(* IEC 61131-3 sources: RL_MAR/experiments/comparison/llm4plc/results/gpt-4o-mini_20260506_100619/20260506_102746, 4 files *)

(* ---- generated_code_iteration_0.st ---- *)
ructured-text
START_ST
FUNCTION_BLOCK FB_SimpleRepeat
VAR_INPUT
    INPUT_VAR1 : INT := 2; // Initial value
    INPUT_COUNTER : INT := 4; // Number of iterations
END_VAR

VAR_OUTPUT
    OUTPUT_VAR1 : INT; // Final computed value
END_VAR

VAR
    COUNTER : INT; // Counter for iterations
    state : INT; // The state variable
END_VAR

// Logic Implementation
state := 0; // Initialize state

REPEAT
    CASE state OF
        0: // STATE 0: INITIALIZE
            OUTPUT_VAR1 := INPUT_VAR1; // Initialize OUTPUT_VAR1
            COUNTER := INPUT_COUNTER; // Set COUNTER to INPUT_COUNTER
            IF COUNTER > 0 THEN
                state := 1; // Transition to STATE 1
            END_IF;

        1: // STATE 1: REPEAT MULTIPLICATION
            OUTPUT_VAR1 := OUTPUT_VAR1 * 2; // Multiply OUTPUT_VAR1 by 2
            COUNTER := COUNTER - 1; // Decrement COUNTER
            IF COUNTER > 0 THEN
                state := 1; // Stay in STATE 1
            ELSE
                state := 0; // Transition back to STATE 0
            END_IF;
    END_CASE;
UNTIL state = 0; // Loop until state is 0
END_FUNCTION_BLOCK
END_ST

(* ---- generated_code_iteration_1.st ---- *)
START_REASON
The errors in the original Structured Text (ST) code occurred due to the incorrect termination of the REPEAT loop. The feedback specifically indicated that the correct syntax requires the use of 'END_REPEAT' instead of a semicolon. This is a critical syntax requirement in Structured Text programming. Therefore, I will correct the termination of the REPEAT loop and ensure that the overall structure adheres to the standards of a FUNCTION_BLOCK.
END_REASON

START_ST
FUNCTION_BLOCK FB_SimpleRepeat
VAR_INPUT
    INPUT_VAR1 : INT := 2; // Initial value
    INPUT_COUNTER : INT := 4; // Number of iterations
END_VAR

VAR_OUTPUT
    OUTPUT_VAR1 : INT; // Final computed value
END_VAR

VAR
    COUNTER : INT; // Counter for iterations
    state : INT; // The state variable
END_VAR

// Logic Implementation
state := 0; // Initialize state

REPEAT
    CASE state OF
        0: // STATE 0: INITIALIZE
            OUTPUT_VAR1 := INPUT_VAR1; // Initialize OUTPUT_VAR1
            COUNTER := INPUT_COUNTER; // Set COUNTER to INPUT_COUNTER
            IF COUNTER > 0 THEN
                state := 1; // Transition to STATE 1
            END_IF;

        1: // STATE 1: REPEAT MULTIPLICATION
            OUTPUT_VAR1 := OUTPUT_VAR1 * 2; // Multiply OUTPUT_VAR1 by 2
            COUNTER := COUNTER - 1; // Decrement COUNTER
            IF COUNTER > 0 THEN
                state := 1; // Stay in STATE 1
            ELSE
                state := 0; // Transition back to STATE 0
            END_IF;
    END_CASE;
UNTIL state = 0; // Loop until state is 0
END_REPEAT; // Correct termination of the REPEAT loop
END_FUNCTION_BLOCK
END_ST

(* ---- generated_code_iteration_2.st ---- *)
START_REASON
The errors in the original Structured Text (ST) code occurred due to the incorrect termination of the REPEAT loop. The feedback specifically indicated that the correct syntax requires the use of 'END_REPEAT' instead of a semicolon. This is a critical syntax requirement in Structured Text programming. Therefore, I will correct the termination of the REPEAT loop and ensure that the overall structure adheres to the standards of a FUNCTION_BLOCK. Additionally, I will ensure that the variable sections are properly closed with 'END_VAR' and maintain the FUNCTION_BLOCK structure as required.
END_REASON

START_ST
FUNCTION_BLOCK FB_SimpleRepeat
VAR_INPUT
    INPUT_VAR1 : INT := 2; // Initial value
    INPUT_COUNTER : INT := 4; // Number of iterations
END_VAR

VAR_OUTPUT
    OUTPUT_VAR1 : INT; // Final computed value
END_VAR

VAR
    COUNTER : INT; // Counter for iterations
    state : INT; // The state variable
END_VAR

// Logic Implementation
state := 0; // Initialize state

REPEAT
    CASE state OF
        0: // STATE 0: INITIALIZE
            OUTPUT_VAR1 := INPUT_VAR1; // Initialize OUTPUT_VAR1
            COUNTER := INPUT_COUNTER; // Set COUNTER to INPUT_COUNTER
            IF COUNTER > 0 THEN
                state := 1; // Transition to STATE 1
            END_IF;

        1: // STATE 1: REPEAT MULTIPLICATION
            OUTPUT_VAR1 := OUTPUT_VAR1 * 2; // Multiply OUTPUT_VAR1 by 2
            COUNTER := COUNTER - 1; // Decrement COUNTER
            IF COUNTER > 0 THEN
                state := 1; // Stay in STATE 1
            ELSE
                state := 0; // Transition back to STATE 0
            END_IF;
    END_CASE;
UNTIL state = 0; // Loop until state is 0
END_REPEAT; // Correct termination of the REPEAT loop
END_FUNCTION_BLOCK
END_ST

(* ---- generated_code_iteration_3.st ---- *)
START_REASON
The errors in the original Structured Text (ST) code were primarily due to the incorrect termination of the REPEAT loop, which should use 'END_REPEAT' instead of a semicolon. Additionally, the variable sections were not properly closed with 'END_VAR', and there was a misunderstanding regarding the structure of the FUNCTION_BLOCK. I will ensure that the REPEAT loop is correctly terminated and that the variable sections are properly structured. The overall code will be reviewed to ensure it adheres to the standards of Structured Text programming.
END_REASON

START_ST
FUNCTION_BLOCK FB_SimpleRepeat
VAR_INPUT
    INPUT_VAR1 : INT := 2; // Initial value
    INPUT_COUNTER : INT := 4; // Number of iterations
END_VAR

VAR_OUTPUT
    OUTPUT_VAR1 : INT; // Final computed value
END_VAR

VAR
    COUNTER : INT; // Counter for iterations
    state : INT; // The state variable
END_VAR

// Logic Implementation
state := 0; // Initialize state

REPEAT
    CASE state OF
        0: // STATE 0: INITIALIZE
            OUTPUT_VAR1 := INPUT_VAR1; // Initialize OUTPUT_VAR1
            COUNTER := INPUT_COUNTER; // Set COUNTER to INPUT_COUNTER
            IF COUNTER > 0 THEN
                state := 1; // Transition to STATE 1
            END_IF;

        1: // STATE 1: REPEAT MULTIPLICATION
            OUTPUT_VAR1 := OUTPUT_VAR1 * 2; // Multiply OUTPUT_VAR1 by 2
            COUNTER := COUNTER - 1; // Decrement COUNTER
            IF COUNTER > 0 THEN
                state := 1; // Stay in STATE 1
            ELSE
                state := 0; // Transition back to STATE 0
            END_IF;
    END_CASE;
UNTIL state = 0; // Loop until state is 0
END_REPEAT; // Correct termination of the REPEAT loop
END_FUNCTION_BLOCK
END_ST
